FUNCTION_BLOCK PumpControl02
VAR_INPUT
	LsLow							:	BOOL;		// limit switch LOW (NO)
	LsMiddle						:	BOOL;		// limit switch MIDDLE (NO)
	LsHigh							:	BOOL;		// limit switch HIGH (NC)
END_VAR
VAR_OUTPUT
	Motor1							:	BOOL;		// motor 1 output
	Motor2							:	BOOL;		// motor 2 output
END_VAR
VAR
	SeqStep							:	(INIT, LOW, MIDDLE, HIGH) := INIT;
	RunMotor						:	BOOL;		// pump alternation control
END_VAR

SeqSelect();
SeqOutput();

METHOD SeqOutput : BOOL
VAR_INPUT
END_VAR

VAR
	StepMiddleOneShot: R_TRIG;
END_VAR
VAR_INST // added by the converter: edge detectors and wires of the graphical bodies
    _w1, _w2, _w3 : BOOL;
END_VAR
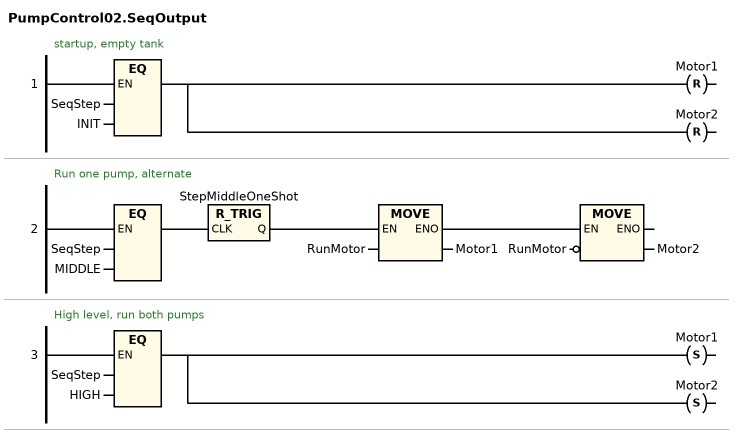
// NETWORK 1
// startup, empty tank
_w1 := SeqStep = INIT;
Motor1 R= _w1;
Motor2 R= _w1;

// NETWORK 2
// Run one pump, alternate
StepMiddleOneShot(CLK := SeqStep = MIDDLE); // R_TRIG
_w2 := StepMiddleOneShot.Q;
IF _w2 THEN Motor1 := RunMotor; END_IF
IF _w2 THEN Motor2 := NOT RunMotor; END_IF

// NETWORK 3
// High level, run both pumps
_w3 := SeqStep = HIGH;
Motor1 S= _w3;
Motor2 S= _w3;
END_METHOD

METHOD SeqSelect : BOOL
VAR_INPUT
END_VAR
VAR_INST // added by the converter: edge detectors and wires of the graphical bodies
    _w1 : BOOL;
END_VAR
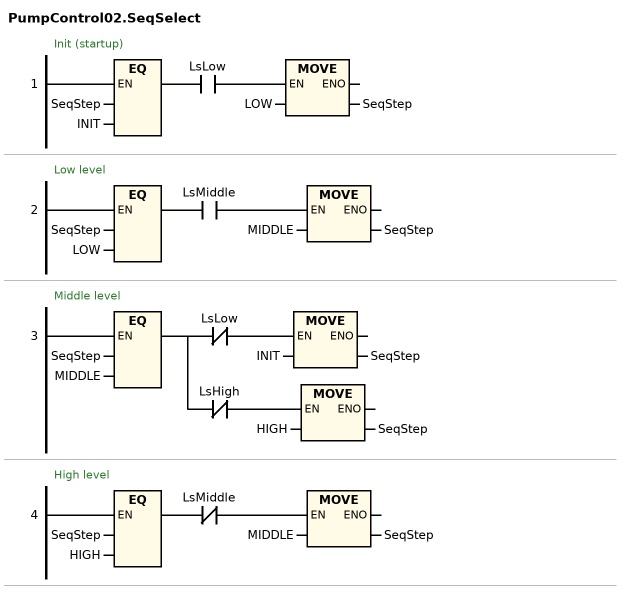
// NETWORK 1
// Init (startup)
IF SeqStep = INIT AND LsLow THEN SeqStep := LOW; END_IF

// NETWORK 2
// Low level
IF SeqStep = LOW AND LsMiddle THEN SeqStep := MIDDLE; END_IF

// NETWORK 3
// Middle level
_w1 := SeqStep = MIDDLE;
IF _w1 AND NOT LsLow THEN SeqStep := INIT; END_IF
IF _w1 AND NOT LsHigh THEN SeqStep := HIGH; END_IF

// NETWORK 4
// High level
IF SeqStep = HIGH AND NOT LsMiddle THEN SeqStep := MIDDLE; END_IF
END_METHOD

END_FUNCTION_BLOCK

(* stored: Version 1.1.0.1, ProductVersion 3.1.4024.15
   POU PumpControl02: Id {3e2fd8b0-db69-4caa-ab32-38d6b745f4a4}, SpecialFunc None
   Method SeqOutput: Id {a2a58b1f-4466-40e2-82fb-2338c2421603}
   Method SeqSelect: Id {96e4813f-0986-4178-8b36-c54ae8a73a5d} *)
